INTERFACE I_RpcReleaseHandle

METHOD ReleaseHandle : ST_AdsStatus
VAR_INPUT
END_VAR
END_METHOD

END_INTERFACE

(* stored: Version 1.1.0.1, ProductVersion 3.1.4024.12
   Itf I_RpcReleaseHandle: Id {bb98d4ca-0a35-4682-8ad6-8c5cd7a7858b}
   Method ReleaseHandle: Id {2bfcaf86-a73b-4e47-95bc-846f7865c600} *)
